# EPICS substitutions: db/Beckhoff_2XXX/ecmcEL2502.substitutions
file "ecmcEcSlave.template"
{
  pattern {}
          {}
}

file "ecmcEL2502-chX.template"
{
  pattern {CH_ID, LINR,    ESLO,            EOFF,    EGU,    PREC, LOW, LOLO, HIGH, HIHI, HYST, LLSV,       LSV,        HSV,        HHSV,     DRVL,  DRVH}
          {1,     "SLOPE", 7.324442274E-4,  0,      "V",     0,    0,   0,    0,    0,    0,    "NO_ALARM", "NO_ALARM", "NO_ALARM", "NO_ALARM", 0,   24}
          {2,     "SLOPE", 7.324442274E-4,  0,      "V",     0,    0,   0,    0,    0,    0,    "NO_ALARM", "NO_ALARM", "NO_ALARM", "NO_ALARM", 0,   24}
}
